TYPE ST_LASER_TEST_SETTINGS :
STRUCT
	height:		UDINT := 20;
	width:		UDINT := 20;
	x:			UDINT := 800;
	y:			UDINT := 900;
	
	threshold:	LREAL := 230;		// Average pixel value for the test to be successfull
END_STRUCT
END_TYPE

(* stored: Version 1.1.0.1
   DUT ST_LASER_TEST_SETTINGS: Id {1974391c-918f-401d-a61a-c351dd2465ed} *)
